(* IEC 61131-3 sources: as-docs/tests/fixtures/SampleProject/Logical/MotorControl, 2 files *)

(* ---- MotorControl.st ---- *)
(*
 * MotorControl FB — Controls motor speed with ramp and fault detection
 *)
FUNCTION_BLOCK MotorControl

R_TRIG_start.CLK := Enable;
R_TRIG_start();

IF Enable THEN
	TON_delay.IN := TRUE;
	TON_delay.PT := T#500ms;
	TON_delay();
	IF TON_delay.Q THEN
		ActualSpeed := SpeedSetpoint;
		Running := TRUE;
	END_IF
ELSE
	TON_delay.IN := FALSE;
	TON_delay();
	ActualSpeed := 0.0;
	Running := FALSE;
END_IF

gMotorSpeed := ActualSpeed;

END_FUNCTION_BLOCK

(* ---- MotorControl.var ---- *)
VAR_INPUT
	Enable      : BOOL;
	SpeedSetpoint : REAL;   (* Speed setpoint [rpm] *)
END_VAR
VAR_OUTPUT
	ActualSpeed : REAL;     (* Measured speed [rpm] *)
	Running     : BOOL;
END_VAR
VAR
	TON_delay   : TON;
	R_TRIG_start : R_TRIG;
END_VAR
